Fanuc KAREL source: NC0054.KL

-- PROVISIONAL review KL for V1013-1; original PC SHA256 bd111cc3b3df855e075aa4268a4e9ed82b25e5480f877da94f2f60d3cd06d58d
-- Incomplete behavior may be omitted. Consult companion uncertainty JSON. Do not deploy.
PROGRAM NC0054
%NOLOCKGROUP
-- UNRESOLVED_LOCAL_POOL 1 cells at code offset 3; source declarations unknown
-- DIRECT_LOCAL_WORD_ACCESS alone does not prove INTEGER, REAL, or BOOLEAN
BEGIN
  -- UNRESOLVED_PC offsets 0-8; opcodes 2B,2C,7B
  -- UNRESOLVED_PC offsets 13-20; opcodes 9D,23
  -- UNRESOLVED_PC offsets 25-42; opcodes 21,40,41,42
  -- UNRESOLVED_PC offsets 47-81; opcodes 21,2E,52,23,7A,40,41,42
  -- UNRESOLVED_PC offsets 86-110; opcodes 21,2E,52,23,7A,43
  -- UNRESOLVED_PC offsets 115-128; opcodes 21,9D,57,79
  -- UNRESOLVED_PC offsets 133-151; opcodes 21,2E,52,23
  -- UNRESOLVED_PC offsets 156-161; opcodes 7A
  -- UNRESOLVED_PC offsets 166-183; opcodes 21,40,41,42
  -- UNRESOLVED_PC offsets 188-222; opcodes 21,2E,52,23,7A,40,41,42
  -- UNRESOLVED_PC offsets 227-251; opcodes 21,2E,52,23,7A,43
  -- UNRESOLVED_PC offsets 256-270; opcodes 21,9D,52,23
  -- UNRESOLVED_PC offsets 290-294; opcodes 7F
  -- UNRESOLVED_PC offsets 299-303; opcodes 27,AA
  -- UNRESOLVED_PC offsets 308-312; opcodes 7F
END NC0054
